(* CODESYS project Magasin Station PLC code.project

Project tree, tasks and I/O mapping:
  Device : CODESYS Control Win V3, 3S - Smart Software Solutions GmbH, order no. 305021, version 3.5.11.30
    application Application
      libraries: Standard, * (System)
      task MainTask (cyclic, interval t#20ms, priority 1) calls PLC_PRG
      program PLC_PRG [LD]
      Symbols
      global variables GVL
*)

// Device/Application/GVL
{attribute 'qualified_only'}
VAR_GLOBAL
	PE_1: BOOL;
	HS2: BOOL;
	HS3: BOOL;
	PE_2: BOOL;
	PE_3: BOOL;
	
	PE1: BOOL;
	PE2: BOOL:=FALSE;
	PE3: BOOL;
	PE4: BOOL;
	
	PEj_1: BOOL;
	PEj_2: BOOL;
	PEj_3: BOOL;
	PEj_4: BOOL;
	
	PInj_1:BOOL;
	PInj_2:BOOL;
	PInj_3:BOOL;
	PInj_4:BOOL;
	
	MF1:BOOL;
	MB1:BOOL;
	MF2: BOOL;
	MB2: BOOL;
	MF3: BOOL;
	MB3: BOOL;
	
	HS1 : BOOL;
	
	stop:BOOL:=TRUE;
	Dump: BOOL;
	start:BOOL;
	ON: BOOL;
	
	MH1: BOOL;
	MH2: BOOL;
	MH3: BOOL;
END_VAR

// Device/Application/PLC_PRG
PROGRAM PLC_PRG
VAR
	

	TON_0: TON;
	TON_1: TON;
	TOF_0: TOF;
	TON_2: TON;
	TON_3: TON;
	F_TRIG_0: F_TRIG;
	F_TRIG_1: F_TRIG;
	F_TRIG_2: F_TRIG;
	FE_PE3: BOOL;
END_VAR

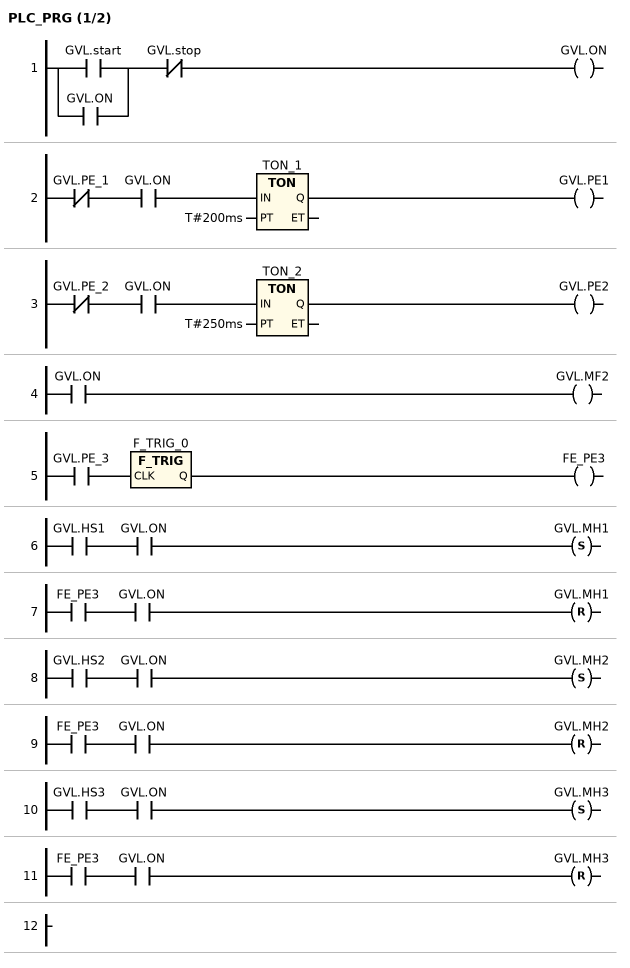
// NETWORK 1
GVL.ON := (GVL.start OR GVL.ON) AND NOT GVL.stop;

// NETWORK 2
TON_1(IN := NOT GVL.PE_1 AND GVL.ON, PT := T#200ms); // TON
GVL.PE1 := TON_1.Q;

// NETWORK 3
TON_2(IN := NOT GVL.PE_2 AND GVL.ON, PT := T#250ms); // TON
GVL.PE2 := TON_2.Q;

// NETWORK 4
GVL.MF2 := GVL.ON;

// NETWORK 5
F_TRIG_0(CLK := GVL.PE_3); // F_TRIG
FE_PE3 := F_TRIG_0.Q;

// NETWORK 6
GVL.MH1 S= GVL.HS1 AND GVL.ON;

// NETWORK 7
GVL.MH1 R= FE_PE3 AND GVL.ON;

// NETWORK 8
GVL.MH2 S= GVL.HS2 AND GVL.ON;

// NETWORK 9
GVL.MH2 R= FE_PE3 AND GVL.ON;

// NETWORK 10
GVL.MH3 S= GVL.HS3 AND GVL.ON;

// NETWORK 11
GVL.MH3 R= FE_PE3 AND GVL.ON;

// NETWORK 12

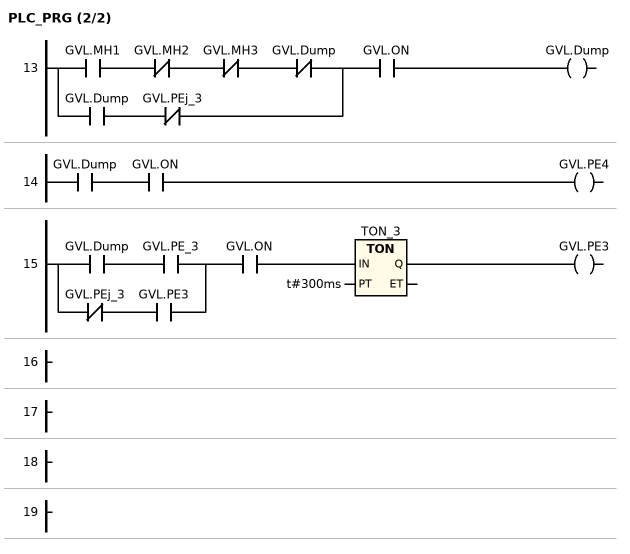
// NETWORK 13
GVL.Dump := (GVL.MH1 AND NOT GVL.MH2 AND NOT GVL.MH3 AND NOT GVL.Dump OR GVL.Dump AND NOT GVL.PEj_3) AND GVL.ON;

// NETWORK 14
GVL.PE4 := GVL.Dump AND GVL.ON;

// NETWORK 15
TON_3(IN := (GVL.Dump AND GVL.PE_3 OR NOT GVL.PEj_3 AND GVL.PE3) AND GVL.ON, PT := t#300ms); // TON
GVL.PE3 := TON_3.Q;

// NETWORK 16

// NETWORK 17

// NETWORK 18

// NETWORK 19

END_PROGRAM
